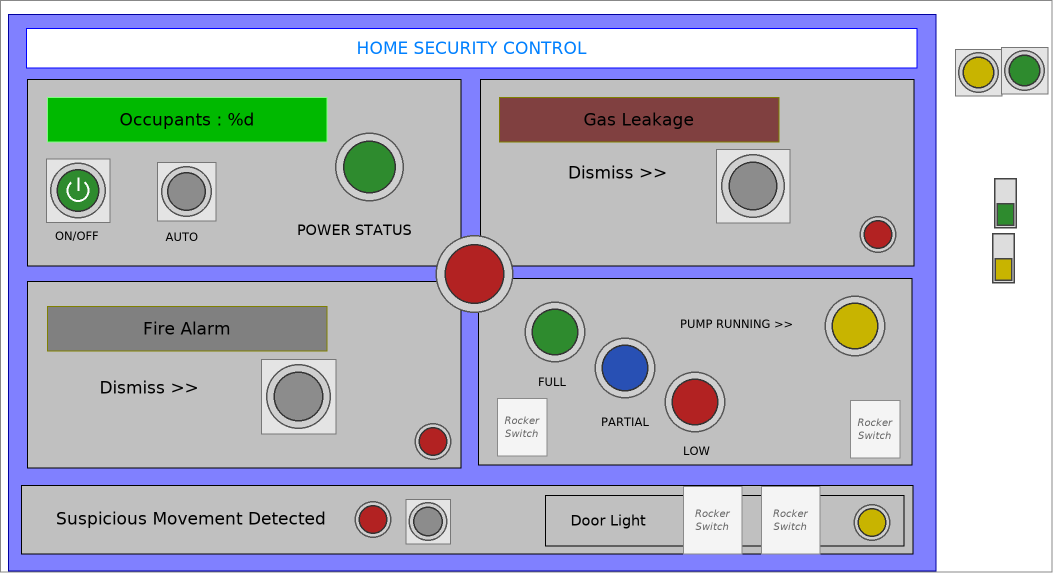
VISUALIZATION Visualization  // 1053x573
    Rectangle (8,14 928x557)
    RoundedRectangle (26,28 891x40), "HOME SECURITY CONTROL"
    RoundedRectangle (21,485 892x69), colour toggle: bSMTlatch
    RoundedRectangle (27,79 434x187)
    RoundedRectangle (480,79 434x187), colour toggle: bMq6latch
    RoundedRectangle (27,281 434x187), colour toggle: bMq2latch
    RoundedRectangle (478,278 434x187)
    Rectangle (47,97 280x45), "Occupants : %d", text variable: iCount
    Rectangle (39,221 76x30), "ON/OFF"
    Rectangle (144,222 76x30), "AUTO"
    PushSwitchLed (157,161 59x61), variable: bAuto, behaviour: TOGGLE, style: Switch-PushSwitchLed-Gray
    Lamp1 (326,127 87x80), variable: bOffOccn, style: Lamp-Lamp1-Green
    Rectangle (282,215 145x30), "POWER STATUS"
    Rectangle (499,97 280x45), "Gas Leakage"
    Rectangle (500,150 235x45), "Dismiss >>", invisible if: Not bMq6latch
    Lamp1 (856,213 44x43), variable: bMq6O, style: Lamp-Lamp1-Red
    Rectangle (47,306 280x45), "Fire Alarm"
    Lamp1 (411,420 44x43), variable: bMq2O, style: Lamp-Lamp1-Red
    Rectangle (47,365 204x45), "Dismiss >>", invisible if: Not bMq2latch
    Lamp1 (520,297 70x70), variable: bFull, style: Lamp-Lamp1-Green
    Lamp1 (590,333 70x70), variable: bPart, style: Lamp-Lamp1-Blue
    Lamp1 (660,367 70x70), variable: bLow, style: Lamp-Lamp1-Red
    Rectangle (514,367 76x30), "FULL"
    Rectangle (587,407 76x30), "PARTIAL"
    Rectangle (659,439 75x24), "LOW"
    Rectangle (36,496 310x45), "Suspicious Movement Detected"
    Lamp1 (351,498 44x43), variable: bSMO, style: Lamp-Lamp1-Red
    RoundedRectangle (545,495 359x51), "Door Light"
    Lamp1 (850,501 44x43), variable: bDLO, style: Lamp-Lamp1-Yellow
    RockerSwitch (683,486 59x68), variable: bDLmanl, behaviour: TOGGLE, style: Switch-RockerSwitch-Green
    PowerSwitch (46,158 64x65), variable: bManl, behaviour: TOGGLE, style: Switch-PowerSwitch-Green
    PushSwitch (952,49 53x47), variable: bI, behaviour: TOGGLE, style: Switch-PushSwitch-Yellow
    PushSwitchLed (401,499 54x45), variable: bSMdismiss, behaviour: TAP, style: Switch-PushSwitchLed-Gray
    PushSwitchLed (256,359 85x75), variable: bMq2dismiss, behaviour: TAP, style: Switch-PushSwitchLed-Gray
    PushSwitchLed (710,149 86x74), variable: bMq6dismiss, behaviour: TAP, style: Switch-PushSwitchLed-Gray
    DipSwitch (979,178 53x50), variable: bH, behaviour: TOGGLE, style: Switch-DipSwitch-Green
    DipSwitch (977,233 53x50), variable: bL, behaviour: TOGGLE, style: Switch-DipSwitch-Yellow
    RockerSwitch (497,398 50x58), variable: bLvlManl, behaviour: TOGGLE, style: Switch-RockerSwitch-Green
    RockerSwitch (850,400 50x58), variable: bLvlManlOff, behaviour: TOGGLE, style: Switch-RockerSwitch-Red
    Lamp1 (427,229 95x90), variable: MAIN.bHazard, style: Lamp-Lamp1-Red
    Lamp1 (820,291 70x70), variable: bTrig, style: Lamp-Lamp1-Yellow
    Rectangle (671,309 131x30), "PUMP RUNNING >>"
    RockerSwitch (761,486 59x68), variable: bDLmanlO, behaviour: TOGGLE, style: Switch-RockerSwitch-Red
    PushSwitch (998,47 53x47), variable: bII, behaviour: TOGGLE, style: Switch-PushSwitch-Green
END_VISUALIZATION

(* stored: Version 1.1.0.1, ProductVersion 3.1.4018.9
   Visu Visualization: Id {5c3e2d85-564c-499b-90e6-8a4361634b5c} *)
